TYPE ST_bit16 :
STRUCT
	A1:BOOL;
	A2:BOOL;
	A3:BOOL;
	A4:BOOL;
	A5:BOOL;
	A6:BOOL;
	A7:BOOL;
	A8:BOOL;
	A9:BOOL;
	A10:BOOL;
	A11:BOOL;
	A12:BOOL;
	A13:BOOL;
	A14:BOOL;
	A15:BOOL;
	A16:BOOL;
END_STRUCT
END_TYPE
